// TIA Portal V20 export
// export: Created 2025-12-01T14:57:04.8399437Z, ExportSetting None, DisplayName Totally Integrated Automation Portal, DisplayVersion V20 Update 3, DisplayName TIA Portal Openness, DisplayVersion V20 Update 3, DisplayName TIA Portal Version Control Interface, DisplayVersion V20 Update 3, DisplayName STEP 7 Professional, DisplayVersion V20 Update 3, DisplayName STEP 7 Safety, DisplayVersion V20 Update 2, DisplayName WinCC Basic/Comfort/Advanced, DisplayVersion V20 Update 3, DisplayName WinCC Professional, DisplayVersion V20 Update 3, DisplayName WinCC Unified, DisplayVersion V20 Update 3
FUNCTION "FC801_JDT01ControlCOM" : Void   // FC801, STL
TITLE = "ControlCOM" - Control de Comunicaciones
{ S7_Optimized_Access := 'FALSE' }
AUTHOR : TRACKING
NAME : 20150129
VERSION : 3.1
// - Contorol y valida el Enlace entre el PLC y el PC
// - Varible: EnlaceCP_OK
// stored: AutoNumber false
   VAR_TEMP
      Temporal : DWord;   // Temporal para el tratamiento de Result 01
      FTCP_MONI_STATUS : Word;
      WTCP_MONI_STATUS : Word;
      FTCP_MONI_MODE : Byte;
      WTCP_MONI_MODE : Byte;
      FTCP_MONI_NDR : Bool;
      FTCP_MONI_ERROR : Bool;
      WTCP_MONI_NDR : Bool;
      WTCP_MONI_ERROR : Bool;
      TMPEnlace_OK : Bool;
   END_VAR
BEGIN

NETWORK
TITLE = Control del Enlace - Puerto 2000
// - Distribución  - Conexion  - Desconesion  - Final    ------------------------------------------------------------------------------------------------------   Control del Enlace - Distribución   --- Si hay que desconetar   --- Si esta conectado
      A     "DB801_JDT01StatusCOM".CNTRL_Reset;  // Si hay que desconectar
      O     "DB801_JDT01StatusCOM".RecJdT_Reset;
      O     "DB801_JDT01StatusCOM".EmiJdT_Reset;
      JC    DesConectar;

      A     "DB801_JDT01StatusCOM".EnlaceCP_OK;  // Si está conectado
      JC    Final;

      JU    Conectar;  // Hay que conectar

// ------------------------------------------------------------------------------------------------------
// Control del Enlace - Conexion
// --- Mirar si hay que activar Flanco
// --- Mirar si hay petición de conexion activa
// --- Llamada de Conexion
// --- Comprobación de la Conexion

Conectar:NOP   0;
      AN    "DB891_VariablesTCP".TCON_JdT_PLC_Busy;
      AN    "DB891_VariablesTCP".TCON_JdT_PLC_Req;
      AN    "DB891_VariablesTCP".TCON_JdT_PLC_Flanco;
      =     "DB891_VariablesTCP".TCON_JdT_PLC_Flanco;  // -- Activar flanco

      A     "DB891_VariablesTCP".TCON_JdT_PLC_Flanco;
      AN    "DB891_VariablesTCP".TCON_JdT_PLC_Req;
      S     "DB891_VariablesTCP".TCON_JdT_PLC_Req;
      R     "DB891_VariablesTCP".TDISCON_JdT_PLC_Req;  // -- Petición de Conexion Activa

      CALL  TCON, "DB892_TCON_JdT_PLC"
      ( REQ     := "DB891_VariablesTCP".TCON_JdT_PLC_Flanco,
        ID      := W#16#1,
        DONE    := "DB891_VariablesTCP".TCON_JdT_PLC_Done,
        BUSY    := "DB891_VariablesTCP".TCON_JdT_PLC_Busy,
        ERROR   := "DB891_VariablesTCP".TCON_JdT_PLC_Error,
        STATUS  := "DB891_VariablesTCP".TCON_JdT_PLC_Status,
        CONNECT := "DB800_JDT01ConfigEnlace"
      );


      A     "DB891_VariablesTCP".TCON_JdT_PLC_Done;  // -- Comprobacion de la Conexion
      R     "DB891_VariablesTCP".TCON_JdT_PLC_Req;
      S     "DB801_JDT01StatusCOM".EnlaceCP_OK;

      A     "DB891_VariablesTCP".TCON_JdT_PLC_Error;  // -- Error en conexion
      R     "DB891_VariablesTCP".TCON_JdT_PLC_Req;

      A     "DB891_VariablesTCP".TCON_JdT_PLC_Req;  // --- Control de Bloqueo
      AN    "DB891_VariablesTCP".TCON_JdT_PLC_Busy;
      R     "DB891_VariablesTCP".TCON_JdT_PLC_Req;

      JU    Final;  // Fin de la Conexión

// ------------------------------------------------------------------------------------------------------
// Control del Enlace - Desconexion
// --- Mirar si hay que activar Flanco
// --- Mirar si hay petición de desconexion activa
// --- Llamada de DesConexion
// --- Comprobación de la DesConexion

DesConectar:SET;
      R     "DB801_JDT01StatusCOM".EnlaceCP_OK;

      AN    "DB891_VariablesTCP".TDISCON_JdT_PLC_Busy;
      AN    "DB891_VariablesTCP".TDISCON_JdT_PLC_Req;
      AN    "DB891_VariablesTCP".TDISCON_JdT_PLC_Flanco;
      =     "DB891_VariablesTCP".TDISCON_JdT_PLC_Flanco;  // -- Activar Flanco

      A     "DB891_VariablesTCP".TDISCON_JdT_PLC_Flanco;
      AN    "DB891_VariablesTCP".TDISCON_JdT_PLC_Req;
      S     "DB891_VariablesTCP".TDISCON_JdT_PLC_Req;
      R     "DB891_VariablesTCP".TCON_JdT_PLC_Req;  // -- Petición de DesConexion Activa

      CALL  TDISCON, "DB893_TDISCON_JdT_PLC"
      ( REQ    := "DB891_VariablesTCP".TDISCON_JdT_PLC_Flanco,
        ID     := W#16#1,
        DONE   := "DB891_VariablesTCP".TDISCON_JdT_PLC_Done,
        BUSY   := "DB891_VariablesTCP".TDISCON_JdT_PLC_Busy,
        ERROR  := "DB891_VariablesTCP".TDISCON_JdT_PLC_Error,
        STATUS := "DB891_VariablesTCP".TDISCON_JdT_PLC_Status
      );

      A     "DB891_VariablesTCP".TDISCON_JdT_PLC_Done;  // -- Comprobacion de la DesConexión
      R     "DB891_VariablesTCP".TDISCON_JdT_PLC_Req;
      R     "DB801_JDT01StatusCOM".CNTRL_Reset;
      R     "DB801_JDT01StatusCOM".RecJdT_Reset;
      R     "DB801_JDT01StatusCOM".EmiJdT_Reset;

      A     "DB891_VariablesTCP".TDISCON_JdT_PLC_Error;  // -- Error en la DesConexion
      R     "DB891_VariablesTCP".TDISCON_JdT_PLC_Req;

      O(;
      L     "DB891_VariablesTCP".TDISCON_JdT_PLC_Status;
      L     W#16#80A3;  //Se está intentando deshacer una conexión no existente
      ==I;
      );
      O(;
      L     "DB891_VariablesTCP".TDISCON_JdT_PLC_Status;
      L     W#16#8086;  //El parámetro ID se encuentra en un rango no permitido
      ==I;
      );
      R     "DB891_VariablesTCP".TDISCON_JdT_PLC_Busy;
      R     "DB891_VariablesTCP".TDISCON_JdT_PLC_Req;
      R     "DB891_VariablesTCP".TDISCON_JdT_PLC_Flanco;

      A     "DB891_VariablesTCP".TDISCON_JdT_PLC_Req;  // --- Control de Bloqueo
      AN    "DB891_VariablesTCP".TDISCON_JdT_PLC_Busy;
      R     "DB891_VariablesTCP".TDISCON_JdT_PLC_Req;

      R     "DB801_JDT01StatusCOM".CNTRL_Reset;
      R     "DB801_JDT01StatusCOM".RecJdT_Reset;
      R     "DB801_JDT01StatusCOM".EmiJdT_Reset;

      JU    Final;  // Fin de la DesConexión

// ------------------------------------------------------------------------------------------------------
// Control del Enlace - Final

Final:NOP   0;


END_FUNCTION
